// Mitsubishi GX Works2 project: 0702-5   PLC: Q02/Q02H

PROGRAM MAIN
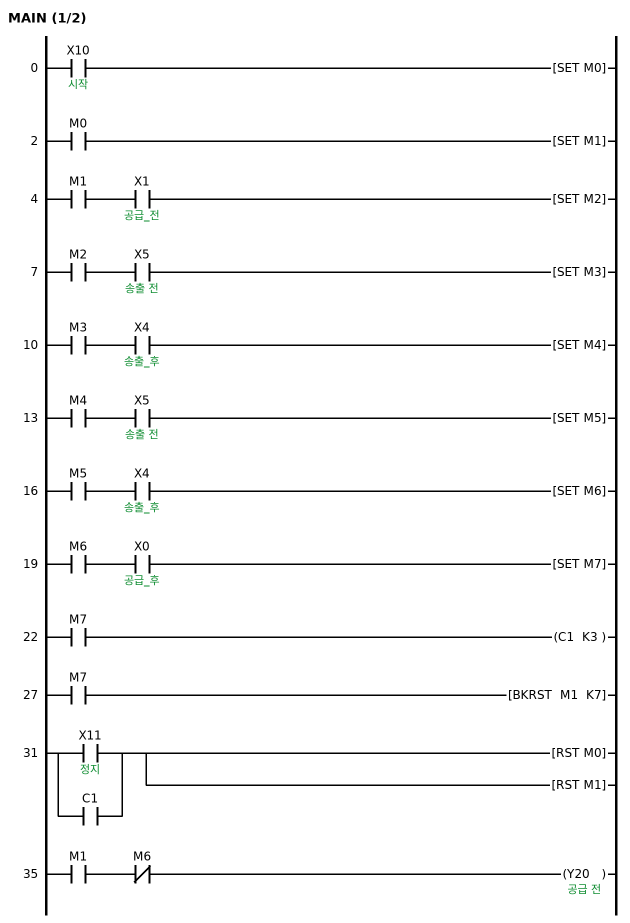
0     LD      X10  ; 시작
      SET     M0
2     LD      M0
      SET     M1
4     LD      M1
      AND     X1  ; 공급_전
      SET     M2
7     LD      M2
      AND     X5  ; 송출 전
      SET     M3
10    LD      M3
      AND     X4  ; 송출_후
      SET     M4
13    LD      M4
      AND     X5  ; 송출 전
      SET     M5
16    LD      M5
      AND     X4  ; 송출_후
      SET     M6
19    LD      M6
      AND     X0  ; 공급_후
      SET     M7
22    LD      M7
      OUT     C1 K3
27    LD      M7
      BKRST   M1 K7
31    LD      X11  ; 정지
      OR      C1
      RST     M0
      RST     M1
35    LD      M1
      ANI     M6
      OUT     Y20  ; 공급 전
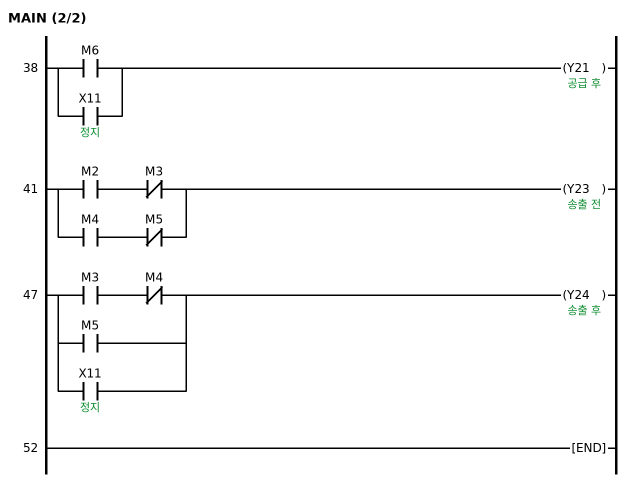
38    LD      M6
      OR      X11  ; 정지
      OUT     Y21  ; 공급 후
41    LD      M2
      ANI     M3
      LD      M4
      ANI     M5
      ORB
      OUT     Y23  ; 송출 전
47    LD      M3
      ANI     M4
      OR      M5
      OR      X11  ; 정지
      OUT     Y24  ; 송출 후
52    END
END_PROGRAM

// device comments not shown above
X2  ; 드릴_상
X3  ; 드릴_하
X6  ; 배출 후
X7  ; 배출 전
Y22  ; 드릴 전
Y25  ; 배출 전
Y26  ; 배출 후
